TYPE ST_HMIWebDriveCommand :
STRUCT
	PowerOn		: BOOL;
	PowerOff	: BOOL;
	Reset		: BOOL;
	Stop 		: BOOL ;
	Calibrate	: BOOL;
	
	SetTension 	: LREAL;
	ScrollDist	: LREAL;
END_STRUCT
END_TYPE

(* stored: Version 1.1.0.1
   DUT ST_HMIWebDriveCommand: Id {24c9034d-f86c-4664-a257-7c0323ce05c2} *)
